Yaskawa INFORM job: R1_W02,4,6(0_0)_KM-OK.JBI

/JOB
//NAME R1_W02,4,6(0_0)_KM-OK
///FOLDERNAME KRIS-SCIANA
//POS
///NPOS 79,79,0,4,0,0
///TOOL 0
///POSTYPE PULSE
///PULSE
C00000=174522,6583,732,81114,57384,11781
C00001=172960,12703,8525,82305,58217,10791
C00002=173420,13658,9390,82287,57878,10798
C00003=172960,12703,8525,82305,58217,10791
C00004=172483,14222,9903,82389,58551,10725
C00005=172960,12703,8525,82305,58217,10791
C00006=174088,5167,5264,84729,55731,9256
C00007=171280,11849,6984,89376,52288,7705
C00008=171280,12128,8246,89869,52259,7340
C00009=171280,11849,6984,89376,52288,7705
C00010=176368,5115,10483,94107,48535,4388
C00011=161133,-21431,-11620,32290,31717,-38951
C00012=166193,-13735,-2683,28322,28551,-36737
C00013=166365,-11916,-1340,28035,28588,-36586
C00014=166193,-13735,-2683,28322,28551,-36737
C00015=166484,-12796,-826,28573,27869,-36854
C00016=166193,-13735,-2683,28322,28551,-36737
C00017=161927,-24594,-12798,32484,31998,-39256
C00018=155155,-6207,-30499,23040,84085,-41474
C00019=187974,16007,-465,74860,68606,73739
C00020=187971,16014,-459,74861,68608,73738
C00021=187970,16017,-457,74861,68609,73738
C00022=188065,16322,-175,74847,68538,73741
C00023=187970,16017,-457,74861,68609,73738
C00024=187982,15993,-478,74858,68601,73740
C00025=188123,15688,-759,74825,68507,73762
C00026=187982,15993,-478,74858,68601,73740
C00027=187982,15995,-476,74858,68601,73740
C00028=188055,16230,-74,74890,68512,73687
C00029=187982,15995,-476,74858,68601,73740
C00030=187983,15992,-479,74858,68601,73740
C00031=185123,16527,-5629,74315,71577,75055
C00032=165643,5472,-22008,57816,82906,32840
C00033=153600,-19645,-23752,41320,66430,-4214
C00034=161010,6792,897,39431,61770,-2600
C00035=161008,6803,906,39432,61771,-2600
C00036=161074,6865,1159,39463,61645,-2620
C00037=161075,4879,-316,39487,61556,-2657
C00038=160508,6816,-113,39396,62494,-2543
C00039=160959,7092,1492,34589,61222,-1662
C00040=157931,14438,8425,38644,65989,-5471
C00041=155353,20308,15528,39705,66096,-6633
C00042=153350,7555,1346,39668,68707,-6522
C00043=174436,-11399,3906,23747,38202,-33405
C00044=174416,-11363,3933,23761,38209,-33414
C00045=155155,-6207,-30499,23040,84085,-41474
C00046=167856,42942,44479,44576,87949,-75494
C00047=174201,39824,30698,44830,89717,-71735
C00048=174202,39772,30629,44830,89729,-71730
C00049=174202,39771,30687,44829,89703,-71742
C00050=173753,38726,28593,44851,90472,-71609
C00051=173790,41778,32604,44829,89804,-71890
C00052=174284,39520,30698,43457,86472,-69264
C00053=174527,39515,30359,43444,86501,-69136
C00054=174346,38585,29600,43450,86582,-69183
C00055=174215,39612,30410,43455,86673,-69209
C00056=163437,11239,19048,64558,76519,-55979
C00057=172451,4154,11436,64150,71153,-54099
C00058=171280,9845,20228,64913,70784,-55366
C00059=171222,10442,21000,64966,70748,-55449
C00060=170248,16174,29758,65704,70306,-56674
C00061=167466,13624,23757,64976,73158,-56067
C00062=174214,39663,30476,43455,86662,-69214
C00063=166320,47562,38864,43573,89751,-71531
C00064=155155,-6207,-30499,23040,84085,-41474
C00065=158532,-24414,-4804,32267,22916,-49173
C00066=162219,-15798,1425,26285,22163,-46063
C00067=160659,-10505,5478,28325,22871,-47138
C00068=172313,-36206,-11141,38952,-3654,-41277
C00069=161098,-12444,3311,27327,23025,-46629
C00070=159658,-10599,5699,29947,23053,-47982
C00071=172547,-36456,-10940,38652,-3952,-41129
C00072=172989,-36590,-9857,36223,-4732,-40014
C00073=176283,-34451,2786,26746,-11679,-35443
C00074=177220,-33568,6334,26181,-13518,-35071
C00075=160661,-10807,5180,25528,18740,-47150
C00076=160656,-10808,5155,25519,18754,-47146
C00077=135615,-20366,-13260,37178,48093,-50762
C00078=15978,-102434,-83816,28834,48298,-44128
BC00000=388510,309469,707895
BC00001=377846,297250,698926
BC00002=377846,297250,698926
BC00003=377846,297250,698926
BC00004=377846,297250,698926
BC00005=377846,297250,698926
BC00006=377173,302368,676412
BC00007=374300,324223,580273
BC00008=374300,324223,580270
BC00009=374300,324223,580273
BC00010=389520,310555,658072
BC00011=302385,369501,846935
BC00012=302385,369501,846935
BC00013=302385,369501,846935
BC00014=302385,369501,846935
BC00015=302385,369501,846935
BC00016=302385,369501,846935
BC00017=303063,366371,858833
BC00018=296594,383677,873629
BC00019=388565,349039,658383
BC00020=383620,354242,647781
BC00021=381641,356323,643541
BC00022=379252,356345,643535
BC00023=381641,356323,643541
BC00024=390370,358132,618560
BC00025=390394,360436,618584
BC00026=390370,358132,618560
BC00027=388386,356954,612189
BC00028=388387,356961,604124
BC00029=388386,356954,612189
BC00030=390364,354873,616429
BC00031=395310,349670,627031
BC00032=359912,361864,715458
BC00033=313394,370704,855255
BC00034=313394,370704,855255
BC00035=307271,367223,843128
BC00036=304895,365871,838419
BC00037=304822,365830,838277
BC00038=304822,365830,838277
BC00039=308544,362355,825419
BC00040=308544,362355,825419
BC00041=308544,362355,825419
BC00042=308544,362355,825419
BC00043=333107,324818,928104
BC00044=333060,324815,1035638
BC00045=296594,383677,873629
BC00046=333324,394588,980736
BC00047=333273,394401,873204
BC00048=330544,400099,857707
BC00049=329453,402378,851509
BC00050=329453,402378,851509
BC00051=329453,402378,851509
BC00052=333744,407726,853540
BC00053=351310,407559,799899
BC00054=351310,407559,799899
BC00055=352593,405391,806169
BC00056=355802,399975,821840
BC00057=355802,399975,821840
BC00058=355802,399975,821840
BC00059=355802,399975,821840
BC00060=355802,399975,821840
BC00061=355802,399975,821840
BC00062=355802,399973,821843
BC00063=355852,400159,929375
BC00064=296594,383677,873629
BC00065=301704,360961,1065666
BC00066=301654,360775,958133
BC00067=294938,357626,948793
BC00068=294960,335870,816430
BC00069=292251,356366,945057
BC00070=292251,356366,945057
BC00071=294960,335870,816430
BC00072=294960,335870,816430
BC00073=294960,335870,816430
BC00074=294960,335870,816430
BC00075=292523,376817,836925
BC00076=299118,380341,845574
BC00077=299169,380527,953107
BC00078=277147,401439,968203
///POSTYPE BASE
///RECTAN
///RCONF 0,0,0,0,1,0,0,0,0,0,0,0,0,0,0,0,0,0,0,0,0,0,0,0
P00006=2.006,1.622,-0.565,0.0000,0.0000,0.0000
P00021=0.073,2.058,-0.109,0.0000,0.0000,0.0000
///RCONF 0,0,0,0,0,0,0,0,0,0,0,0,0,0,0,0,0,0,0,0,0,0,0,0
P00024=-1.466,-0.226,-0.419,0.0000,0.0000,0.0000
P00026=2.644,0.055,-2.583,0.0000,0.0000,0.0000
//INST
///DATE 2025/04/11 10:11
///ATTR SC,RW
///GROUP1 RB1,BS1
NOP
SFTOF
MOVL C00000 BC00000 V=333.3
MOVL C00001 BC00001 V=166.7
REFP 3 C00002 BC00002
CALL JOB:SEARCH-R1
SET P021 P006
SFTON P021
MOVL C00003 BC00003 V=60.0
REFP 3 C00004 BC00004
CALL JOB:SEARCH-R1
SET P021 P006
SFTON P021
MOVL C00005 BC00005 V=166.7
MOVL C00006 BC00006 V=166.7
MOVL C00007 BC00007 V=166.7
REFP 3 C00008 BC00008
CALL JOB:SEARCH-R1
SET P021 P006
SFTON P021
MOVL C00009 BC00009 V=166.7
MOVL C00010 BC00010 V=100.0
SFTOF
MOVL C00011 BC00011 V=166.7
MOVL C00012 BC00012 V=166.7
REFP 3 C00013 BC00013
CALL JOB:SEARCH-R1
SET P026 P006
SFTON P026
MOVL C00014 BC00014 V=60.0
REFP 3 C00015 BC00015
CALL JOB:SEARCH-R1
SET P026 P006
SFTON P026
MOVL C00016 BC00016 V=60.0
MOVL C00017 BC00017 V=250.0
MOVJ C00018 BC00018 VJ=100.00
'Path S705 (for W3)
SFTOF
MOVL C00019 BC00019 V=166.7
MOVL C00020 BC00020 V=250.0
MOVL C00021 BC00021 V=250.0
REFP 3 C00022 BC00022
CALL JOB:SEARCH-R1
SET P024 P006
SFTON P024
MOVL C00023 BC00023 V=166.7
MOVL C00024 BC00024 V=166.7
REFP 3 C00025 BC00025
CALL JOB:SEARCH-R1
SET P024 P006
SFTON P024
MOVL C00026 BC00026 V=166.7
MOVL C00027 BC00027 V=166.7
REFP 3 C00028 BC00028
CALL JOB:SEARCH-R1
SET P024 P006
SFTON P024
MOVL C00029 BC00029 V=166.7
MOVL C00030 BC00030 V=166.7
MOVL C00031 BC00031 V=166.7
MOVJ C00032 BC00032 VJ=100.00
MOVJ C00033 BC00033 VJ=100.00
'Path W1
SFTOF
CALL JOB:COFNIJ_DRUT
SFTON P026
MOVL C00034 BC00034 V=166.7
MOVL C00035 BC00035 V=166.7
MOVL C00036 BC00036 V=166.7 PL=0
REFP 1 C00037 BC00037
REFP 2 C00038 BC00038
MACRO1 MJ#(0) ARGF10
ARCON
MOVL C00039 BC00039 V=13.3
MOVL C00040 BC00040 V=13.3
MOVL C00041 BC00041 V=13.3
ARCOF
SFTOF
MOVL C00042 BC00042 V=250.0
'Path W2
SFTOF
SFTON P021
MOVL C00043 BC00043 V=250.0
MOVL C00044 BC00044 V=250.0
SFTOF
'
MOVJ C00045 BC00045 VJ=100.00
'Path W786
SFTOF
SFTON P024
MOVJ C00046 BC00046 VJ=100.00
MOVL C00047 BC00047 V=250.0
MOVL C00048 BC00048 V=166.7
MOVL C00049 BC00049 V=166.7 PL=0
REFP 1 C00050 BC00050
REFP 2 C00051 BC00051
MACRO1 MJ#(0) ARGF10
ARCON
MOVL C00052 BC00052 V=13.3
MOVL C00053 BC00053 V=13.3
MOVL C00054 BC00054 V=11.7
ARCOF
MOVL C00055 BC00055 V=166.7
SFTOF
MOVL C00056 BC00056 V=166.7
MACRO1 MJ#(0) ARGF7
MOVL C00057 BC00057 V=166.7
ARCON
MOVL C00058 BC00058 V=11.7
MOVL C00059 BC00059 V=11.7
MOVL C00060 BC00060 V=11.7
ARCOF
MOVL C00061 BC00061 V=166.7
MOVL C00062 BC00062 V=250.0
MOVL C00063 BC00063 V=250.0
SFTOF
MOVJ C00064 BC00064 VJ=100.00
'
'Path W4
SFTOF
SFTON P021
MOVJ C00065 BC00065 VJ=100.00
MOVL C00066 BC00066 V=333.3
MOVL C00067 BC00067 V=250.0
MOVL C00068 BC00068 V=166.7 PL=0
REFP 1 C00069 BC00069
REFP 2 C00070 BC00070
MACRO1 MJ#(0) ARGF10
ARCON
MOVL C00071 BC00071 V=13.3
MOVL C00072 BC00072 V=13.3
MOVL C00073 BC00073 V=13.3
MOVL C00074 BC00074 V=13.3
ARCOF
MOVL C00075 BC00075 V=166.7
MOVL C00076 BC00076 V=250.0
MOVJ C00077 BC00077 VJ=100.00
MOVJ C00078 BC00078 VJ=100.00
SFTOF
END
